// TIA Portal V19 export
DATA_BLOCK "PPrgArchive9"   // DB505
// stored: IsOnlyStoredInLoadMemory true, MemoryReserve 0, Namespace G
   VAR RETAIN
      PRG : Array[801..900] of "PPrg_Data";
   END_VAR
BEGIN
END_DATA_BLOCK
